INTERFACE IPrinter

METHOD print
VAR_INPUT
END_VAR
END_METHOD

END_INTERFACE

(* stored: Version 1.1.0.1, ProductVersion 3.1.4022.7
   Itf IPrinter: Id {25c20b41-14da-4791-9709-036fa15c27d1}
   Method print: Id {f560a1af-f6e3-43e3-b12a-48a42ee41636} *)
